Universal Robots PolyScope program: MixerPickupLocal.urp

Program MixerPickupLocal (installation=Youssef directory=/programs/Youssef createdIn=5.9.5.1031259 lastSavedIn=5.9.5.1031259 robotSerialNumber=20215500597)
Calibrated DH parameters: a=[0.000193, -0.066673, -0.391568, -0.000012, 0.00005, 0]; d=[0.162643, -472.05677, 465.132521, 7.058239, 0.099746, 0.099582]; alpha=[1.571116, 0.00089, 0.003862, 1.569269, -1.569248, 0]; deltaTheta=[0, -1.413394, 7.628392, 0.068187, 0, -0.000001]
Robot Program (runOnlyOnce=true)
  URCap Gripper (Robotiq_Grippers, Robotiq Inc.) dataModel(position=100.0, force=49.80392156862745, speed=20.0, positionInDouble=100.0, forceInDouble=49.80392156862745, speedInDouble=20.0, slaveIds=[9], blocking=true)
  MoveJ speed 60 deg/s, acceleration 80 deg/s^2 (useActiveTCP=true) feature=Base
    Waypoint Waypoint (Variable): variable(featureName=Mixer_Intact)
    Waypoint Waypoint (Variable): variable(featureName=Mixer_Standby)
  MoveJ speed 60 deg/s, acceleration 80 deg/s^2 (useActiveTCP=true) feature=Base
    Waypoint Waypoint_9: TCP in base x=618.275 y=219.993 z=160.974 mm, rx=1.209 ry=1.2027 rz=1.1964 rad; joints [54.155, -107.639, -124.058, -128.368, -34.984, -0.179] deg; TCP offset x=0 y=0 z=191.5 mm, rx=0 ry=0 rz=0 rad
    Waypoint Waypoint (Variable): variable(featureName=Pickup)
    URCap Gripper (Robotiq_Grippers, Robotiq Inc.) dataModel(position=0.0, force=49.80392156862745, speed=20.0, positionInDouble=0.0, forceInDouble=49.80392156862745, speedInDouble=20.0, slaveIds=[9], blocking=true)
    Waypoint Waypoint (Variable): variable(featureName=Local)
